FUNCTION Extension : INT
VAR_INPUT
	EndPosition: INT;
	State: INT;
END_VAR
VAR
	MovementEnum: Movement;
	NextState: INT;
	MotorDirectionEnum: MovementDirection;
END_VAR

IF Automatic.ExtensionPositionAuto > EndPosition THEN
	MotorDirectionEnum := MovementDirection.TowardsSensor;
ELSE
	MotorDirectionEnum := MovementDirection.AwayFromSensor;
END_IF

IF MotorDirectionEnum = MovementDirection.TowardsSensor THEN
	IF Automatic.ExtensionPositionAuto > EndPosition THEN	// it drops wood in the nearest bin
		IO.MotorExtensionDirection := (MotorDirectionEnum = MovementDirection.TowardsSensor);
		IF NOT Automatic.SafetyEON THEN
			Automatic.ECurrentlyMoving := TRUE;
			IO.MotorExtension := (MovementEnum = Movement.ON);
		END_IF
		NextState := State;
	ELSE
		IO.MotorExtension := (MovementEnum = Movement.OFF);
		NextState := State + 1;
		Automatic.ECurrentlyMoving := FALSE;
	END_IF
ELSE
	IF Automatic.ExtensionPositionAuto < EndPosition THEN
		IO.MotorExtensionDirection := (MotorDirectionEnum = MovementDirection.AwayFromSensor);
		IF NOT Automatic.SafetyEON THEN
			Automatic.ECurrentlyMoving := TRUE;
			IO.MotorExtension := (MovementEnum = Movement.ON);
		END_IF
		NextState := State;
	ELSE
		IO.MotorExtension := (MovementEnum = Movement.OFF);
		NextState := State + 1;
		Automatic.ECurrentlyMoving := FALSE;
	END_IF
END_IF

Extension := NextState;
RETURN;

END_FUNCTION

(* stored: Version 1.1.0.1, ProductVersion 3.1.4024.13
   POU Extension: Id {e06cc85d-8666-43e0-8088-edc0359ce657}, SpecialFunc None *)
